Yaskawa INFORM job: SKRZYNIA_5040_0_STOPNI_2OBR.JBI

/JOB
//NAME SKRZYNIA_5040_0_STOPNI_2OBR
///FOLDERNAME 02-SKRZYNIE_JOBS
//POS
///NPOS 486,486,0,40,0,0
///TOOL 0
///POSTYPE PULSE
///PULSE
C00000=1055,-24125,84372,288,19725,204
C00001=0,-15438,65714,0,-68532,0
C00002=4718,-16587,59952,3396,-65485,-935
C00003=32997,-21499,42555,27623,-61436,21376
C00004=31759,-20688,42932,26837,-60850,21559
C00005=28987,-21156,42712,24818,-60442,22222
C00006=33447,-21964,42352,27886,-61721,21330
C00007=37687,-23357,41794,30651,-63289,20620
C00008=38979,-19018,48057,32961,-64962,20678
C00009=37261,-18075,48526,31902,-64209,20901
C00010=35830,-17198,48994,31015,-63571,21092
C00011=34080,-17614,48768,29780,-63290,21485
C00012=37261,-18075,48526,31902,-64209,20901
C00013=47373,-21912,40596,41149,-66086,26950
C00014=4718,-16587,59952,3396,-65485,-935
C00015=9265,-17323,54007,6858,-62132,-2051
C00016=8830,-16324,54489,6560,-61693,-1980
C00017=6020,-16550,54375,4472,-61664,-1348
C00018=9265,-17323,54007,6858,-62132,-2051
C00019=9252,-17290,54021,6848,-62117,-2048
C00020=9252,-17290,54021,6848,-62117,-2048
C00021=8694,-15983,54664,6467,-61548,-1957
C00022=4418,-16236,54535,3285,-61485,-993
C00023=9252,-17290,54021,6848,-62117,-2048
C00024=8708,-18333,53563,6422,-62559,-1899
C00025=8708,-18333,53563,6422,-62559,-1899
C00026=7766,-16032,54635,5782,-61526,-1748
C00027=5536,-16243,54528,4122,-61523,-1244
C00028=8708,-18333,53563,6422,-62559,-1899
C00029=8708,-18333,53563,6422,-62559,-1899
C00030=8708,-18331,53563,6422,-62556,-1899
C00031=7758,-16002,54651,5775,-61511,-1746
C00032=4943,-16221,54537,3680,-61495,-1109
C00033=30098,-19369,49260,26650,-63246,1300
C00034=73517,-47200,-15425,81407,-61841,11109
C00035=59944,-42786,-13955,78333,-53158,10478
C00036=57437,-41828,-13292,77672,-51559,10479
C00037=55365,-40827,-12885,77319,-50190,10340
C00038=53830,-41542,-13178,76508,-49301,10646
C00039=57437,-41828,-13292,77672,-51559,10479
C00040=52398,-46622,-9296,62308,-52824,5916
C00041=23564,-39822,17337,24809,-47524,-9372
C00042=10104,-46603,4759,11228,-37390,-5046
C00043=0,-52280,40443,0,6876,0
C00044=1529,-42140,58025,-5964,2417,3265
C00045=0,-52280,-4943,-1861,-42535,447
C00046=2621,-57340,-29475,1206,-23680,-711
C00047=2621,-57340,-29475,1206,-23680,-711
C00048=2622,-57337,-29476,1207,-23680,-710
C00049=2506,-56325,-29286,1041,-23045,-642
C00050=-1228,-56520,-29324,-5243,-23254,2072
C00051=2622,-57337,-29476,1207,-23680,-710
C00052=3066,-60430,-29907,1796,-25718,-952
C00053=3066,-47126,-4537,1796,-25717,-952
C00054=1150,-46289,-4389,-1134,-25181,209
C00055=1064,-44762,-4067,-1313,-24253,286
C00056=-2289,-44921,-4103,-6642,-24487,2426
C00057=-2440,-47252,-5097,-6576,-25720,2369
C00058=2574,-52173,738,1108,-22518,-664
C00059=2573,-58294,-29633,1093,-24294,-659
C00060=2321,-56024,-29231,725,-22860,-505
C00061=-1822,-56214,-29269,-6293,-23108,2531
C00062=2573,-58294,-29633,1093,-24294,-659
C00063=26763,-41451,10217,33856,-29391,24493
C00064=43270,-28616,24993,58998,-40730,16959
C00065=40951,-27396,25513,57868,-39388,17043
C00066=39074,-27880,25300,56233,-38652,17553
C00067=43270,-28616,24993,58998,-40730,16959
C00068=49158,-38250,8479,66986,-41880,13443
C00069=1817,-44984,2816,-3462,-45659,1296
C00070=1148,-56354,34370,-22,3827,-10
C00071=0,-52280,40443,0,6876,0
C00072=0,-52280,40443,0,-64237,0
C00073=12053,-46193,863,14693,-33250,-5548
C00074=7764,-43650,5766,9193,-34179,-3413
C00075=6226,-39841,6502,7870,-31713,-3015
C00076=3343,-40039,6452,4230,-31654,-1619
C00077=7764,-43650,5766,9193,-34179,-3413
C00078=7764,-43650,5766,9193,-34179,-3413
C00079=12053,-46193,863,14693,-33250,-5548
C00080=0,-52280,40443,0,6876,0
C00081=0,-52280,40443,0,6876,0
C00082=0,-52280,40443,0,6876,0
C00083=33629,-57276,-6399,46271,-24969,-2804
C00084=75493,-63502,-64712,103874,-64610,-6298
C00085=47077,-58045,-62565,110120,-45736,-10942
C00086=43793,-59800,-66982,115317,-43706,-9888
C00087=62671,-64213,-64640,104431,-56093,-7372
C00088=62671,-64213,-64640,104431,-56093,-7372
C00089=28458,-50318,6850,47420,-25887,-3347
C00090=0,-52280,40443,0,6876,0
C00091=1055,-24125,84372,288,19725,204
C00092=0,-15438,65714,0,-68532,0
C00093=0,-15438,65714,966,-70097,42926
C00094=69988,-9219,57065,61610,-82752,27767
C00095=63113,-6157,59685,58080,-79692,28271
C00096=45688,-7238,64427,40079,-74101,29444
C00097=49853,-5945,65929,43750,-75729,29302
C00098=63113,-6157,59685,58080,-79692,28271
C00099=69988,-9219,57065,61610,-82752,27767
C00100=0,-15438,65714,966,-70097,42926
C00101=0,-15438,65714,0,-68532,0
C00102=1055,-24125,84372,288,19725,204
C00103=0,-52280,40443,0,6876,0
C00104=0,-52280,40443,0,6876,0
C00105=0,-17525,61946,0,273,32004
C00106=54446,-4421,37881,-48560,57645,57448
C00107=45059,-5790,38757,-53071,45868,54447
C00108=47158,-5256,55782,-85306,41004,71351
C00109=33649,8804,54222,-37726,47106,40629
C00110=39487,-20381,-13316,-29947,69517,34787
C00111=45059,-5790,38757,-53071,45868,54447
C00112=54446,-4421,37881,-48560,57645,57448
C00113=0,-17525,61946,0,273,32004
C00114=0,-52280,40443,0,6876,0
C00115=0,-38538,66749,0,-898,0
C00116=0,-52280,40443,0,-79033,35417
C00117=46775,-35113,22190,42926,-67531,20697
C00118=52587,-26056,25345,47610,-66542,17970
C00119=45955,-25207,25003,44102,-63302,18882
C00120=46479,-26455,22189,44748,-62817,18409
C00121=53914,-29436,22058,48262,-67266,17843
C00122=46775,-35113,22190,42926,-67531,20697
C00123=0,-52280,40443,0,-79033,35417
C00124=0,-52280,40443,0,-61239,28081
C00125=53819,-14110,13758,-46164,60155,50576
C00126=48398,-14119,9451,-44868,59619,48162
C00127=40831,-18219,20924,-60631,39508,52867
C00128=25168,-7888,23888,-27338,44347,31248
C00129=48398,-14119,9451,-44868,59619,48162
C00130=63113,-6157,59685,58080,-79692,28271
C00131=47789,-6280,67353,41142,-75661,29541
C00132=46856,-5642,67903,40595,-75324,29647
C00133=49398,-5231,67705,43314,-76061,29572
C00134=31009,-27517,39857,26049,-56286,31820
C00135=0,-52280,40443,0,-61239,28081
C00136=0,-52280,40443,0,6876,0
C00137=0,-52280,40443,0,6876,0
C00138=-99253,-13690,44082,59847,13407,-31313
C00139=-87814,-12734,20141,45739,-14352,-64418
C00140=-86669,-6582,30812,41148,-16781,-62025
C00141=-85055,-5827,31548,44003,-17420,-63187
C00142=-85971,-6262,31124,42409,-17052,-62539
C00143=-86650,-5303,32069,41395,-16716,-62141
C00144=-94954,-14494,-1860,-7818,15857,-59130
C00145=-94509,-5779,9349,-537,24388,-60626
C00146=-94509,-4687,12787,-574,22838,-60605
C00147=-87106,-8124,29339,40061,-16711,-61555
C00148=-85732,-21202,11427,30682,-24763,-59235
C00149=-84150,-10929,23786,31981,-25941,-59678
C00150=-83036,-10419,24246,33504,-26268,-60308
C00151=-84150,-10929,23786,31981,-25941,-59678
C00152=-85291,-9507,25078,30650,-25411,-59154
C00153=-84150,-10929,23786,31981,-25941,-59678
C00154=-85786,-16909,14677,31743,-23900,-59790
C00155=-84150,-10498,24888,31517,-26306,-59436
C00156=-83174,-10052,25293,32841,-26587,-59984
C00157=-84150,-10498,24888,31517,-26306,-59436
C00158=-85258,-9112,26156,30226,-25800,-58928
C00159=-84150,-10498,24888,31517,-26306,-59436
C00160=-87841,-18519,13420,28367,-23534,-58339
C00161=-84150,-10465,24972,31484,-26336,-59417
C00162=-83241,-10052,25348,32714,-26598,-59924
C00163=-84150,-10465,24972,31484,-26336,-59417
C00164=-85145,-9228,26102,30329,-25881,-58963
C00165=-84150,-10465,24972,31484,-26336,-59417
C00166=-86371,-18277,13606,30568,-23951,-59265
C00167=-84345,-11688,21985,32461,-25312,-59957
C00168=-83211,-11173,22442,34044,-25650,-60618
C00169=-84345,-11688,21985,32461,-25312,-59957
C00170=-85283,-10526,23025,31366,-24861,-59525
C00171=-84345,-11688,21985,32461,-25312,-59957
C00172=-86191,-19647,12567,30467,-24278,-59187
C00173=-84345,-10877,24073,31552,-26006,-59481
C00174=-83051,-10286,24607,33321,-26381,-60213
C00175=-84345,-10877,24073,31552,-26006,-59481
C00176=-85179,-9842,25009,30582,-25619,-59100
C00177=-84345,-10877,24073,31552,-26006,-59481
C00178=-85438,-18022,14839,31140,-24818,-59429
C00179=-84247,-11820,22550,32049,-25753,-59727
C00180=-84104,-10976,23642,32111,-25899,-59738
C00181=-82990,-10465,24105,33639,-26227,-60372
C00182=-84104,-10976,23642,32111,-25899,-59738
C00183=-84898,-9998,24525,31196,-25529,-59378
C00184=-84104,-10976,23642,32111,-25899,-59738
C00185=-86610,-16845,14732,30573,-23614,-59301
C00186=-84104,-10864,23927,31990,-25993,-59674
C00187=-82824,-10273,24459,33737,-26370,-60397
C00188=-84104,-10864,23927,31990,-25993,-59674
C00189=-84789,-10021,24690,31200,-25673,-59363
C00190=-84104,-10864,23927,31990,-25993,-59674
C00191=-83806,-19585,12613,33764,-25080,-60559
C00192=-83924,-10205,25475,31619,-26533,-59453
C00193=-82780,-9675,25960,33156,-26866,-60087
C00194=-83924,-10205,25475,31619,-26533,-59453
C00195=-84478,-9530,26093,30986,-26280,-59206
C00196=-83924,-10205,25475,31619,-26533,-59453
C00197=-87149,-17993,13826,29513,-23647,-58830
C00198=-84920,-13182,20975,31162,-25481,-59361
C00199=-83711,-10572,24852,32056,-26475,-59649
C00200=-82779,-10142,25241,33309,-26748,-60166
C00201=-83711,-10572,24852,32056,-26475,-59649
C00202=-84370,-9774,25579,31305,-26170,-59356
C00203=-83711,-10572,24852,32056,-26475,-59649
C00204=-83642,-3679,42021,23358,-36761,-56118
C00205=-85886,-5975,41264,18964,-40261,-54782
C00206=-83919,-11632,22322,32811,-25616,-60079
C00207=-82884,-11162,22742,34234,-25925,-60671
C00208=-83919,-11632,22322,32811,-25616,-60079
C00209=-84723,-10654,23196,31887,-25230,-59715
C00210=-83919,-11632,22322,32811,-25616,-60079
C00211=-87348,-16035,7353,17528,-35245,-56477
C00212=-86244,-15062,8172,18754,-35315,-57058
C00213=-86244,-16649,3638,19674,-33501,-57585
C00214=-85308,-16228,3988,20718,-33648,-58082
C00215=-86244,-16649,3638,19674,-33501,-57585
C00216=-86740,-15973,4201,19194,-33277,-57362
C00217=-86244,-16649,3638,19674,-33501,-57585
C00218=-73780,-8639,20128,34258,-51705,-52097
C00219=-90711,-17528,-28778,11328,-28245,-57111
C00220=-92565,-19610,-33223,7138,-24591,-57051
C00221=-91512,-19116,-32812,8551,-24603,-57834
C00222=-92565,-19610,-33223,7138,-24591,-57051
C00223=-93003,-18716,-32476,6600,-24397,-56752
C00224=-92565,-19610,-33223,7138,-24591,-57051
C00225=-92565,-19610,-33223,7138,-24591,-57051
C00226=-95836,-54375,-51122,6031,-17685,-48210
C00227=-95836,-54375,-51122,6031,-17685,-48210
C00228=-43821,-47238,-2775,-3022,56549,-3681
C00229=-20126,-26882,59542,2406,16879,-9162
C00230=-20126,-26882,59542,2406,16879,-9162
C00231=98601,-10520,92678,4674,-40855,-9615
C00232=95537,-19831,-2695,-2933,-44471,35837
C00233=92548,-20391,-28429,-6186,-30623,55200
C00234=91429,-17018,-28974,-8057,-27827,56250
C00235=91429,-17018,-28974,-8057,-27827,56250
C00236=90371,-16495,-28521,-9286,-27856,56953
C00237=91429,-17018,-28974,-8057,-27827,56250
C00238=92033,-15799,-27911,-7415,-27588,55880
C00239=91429,-17018,-28974,-8057,-27827,56250
C00240=92548,-20391,-28429,-6186,-30623,55200
C00241=91156,-15018,-4648,-8036,-38181,54813
C00242=90585,-14766,-4428,-8565,-38201,55100
C00243=88830,-13959,-3717,-10186,-38284,55977
C00244=89897,-14456,-4157,-9202,-38230,55445
C00245=90761,-12944,-2809,-8452,-37927,55043
C00246=89897,-14456,-4157,-9202,-38230,55445
C00247=89910,-11217,67535,-9455,-58896,55399
C00248=89655,-8493,73265,-9548,-61393,54478
C00249=89910,-11217,67535,-9455,-58896,55399
C00250=85786,-16735,14816,-31782,-23869,59812
C00251=83514,-12996,17929,-35760,-24132,61552
C00252=82251,-12406,18443,-37550,-24551,62308
C00253=83514,-12996,17929,-35760,-24132,61552
C00254=84258,-12095,18717,-34917,-23742,61217
C00255=83514,-12996,17929,-35760,-24132,61552
C00256=87149,-17993,13826,-29513,-23647,58830
C00257=83118,-12818,18089,-36330,-24263,61791
C00258=81915,-12248,18589,-38020,-24666,62504
C00259=83118,-12818,18089,-36330,-24263,61791
C00260=83897,-11882,18912,-35460,-23856,61445
C00261=83118,-12818,18089,-36330,-24263,61791
C00262=83806,-19585,12613,-33764,-25080,60559
C00263=82998,-13006,17925,-36445,-24332,61826
C00264=81675,-12378,18472,-38297,-24777,62607
C00265=82998,-13006,17925,-36445,-24332,61826
C00266=83876,-11958,18841,-35466,-23874,61442
C00267=82998,-13006,17925,-36445,-24332,61826
C00268=86610,-16845,14732,-30573,-23614,59301
C00269=82493,-13239,17725,-37070,-24559,62089
C00270=81406,-12724,18174,-38578,-24928,62723
C00271=82493,-13239,17725,-37070,-24559,62089
C00272=83436,-12134,18690,-36041,-24064,61684
C00273=82493,-13239,17725,-37070,-24559,62089
C00274=84814,-16043,15376,-33312,-24093,60464
C00275=82555,-13613,17404,-36910,-24580,62015
C00276=81384,-13062,17878,-38534,-24974,62698
C00277=82555,-13613,17404,-36910,-24580,62015
C00278=83566,-12434,18427,-35805,-24047,61580
C00279=82555,-13613,17404,-36910,-24580,62015
C00280=86191,-19647,12567,-30467,-24278,59187
C00281=82500,-13648,17375,-36975,-24607,62039
C00282=81467,-13161,17792,-38413,-24955,62645
C00283=82500,-13648,17375,-36975,-24607,62039
C00284=83481,-12505,18364,-35905,-24087,61617
C00285=82500,-13648,17375,-36975,-24607,62039
C00286=86371,-18277,13606,-30568,-23951,59265
C00287=82904,-13790,17251,-36416,-24470,61808
C00288=81715,-13237,17726,-38081,-24865,62509
C00289=82904,-13790,17251,-36416,-24470,61808
C00290=83686,-12878,18037,-35556,-24055,61469
C00291=82904,-13790,17251,-36416,-24470,61808
C00292=87841,-18519,13420,-28367,-23534,58339
C00293=82748,-13879,17174,-36603,-24542,61883
C00294=81692,-13388,17594,-38077,-24893,62505
C00295=82748,-13879,17174,-36603,-24542,61883
C00296=83607,-12881,18032,-35663,-24082,61515
C00297=82748,-13879,17174,-36603,-24542,61883
C00298=85786,-16909,14677,-31743,-23900,59790
C00299=82520,-14198,16902,-36833,-24674,61972
C00300=81460,-13708,17319,-38301,-25026,62591
C00301=82520,-14198,16902,-36833,-24674,61972
C00302=83571,-12989,17938,-35691,-24113,61524
C00303=82520,-14198,16902,-36833,-24674,61972
C00304=85732,-21202,11427,-30682,-24763,59235
C00305=82398,-14365,16763,-36952,-24745,62014
C00306=81172,-13798,17245,-38643,-25153,62725
C00307=82398,-14365,16763,-36952,-24745,62014
C00308=83600,-12984,17944,-35650,-24102,61504
C00309=82398,-14365,16763,-36952,-24745,62014
C00310=83143,-16385,15097,-35497,-24760,61361
C00311=86140,-12802,12665,-93523,-10743,85795
C00312=85030,-12289,13120,-93723,-11463,85776
C00313=86140,-12802,12665,-93523,-10743,85795
C00314=86958,-11660,13681,-94506,-10238,86349
C00315=87761,-14801,10937,-92035,-9671,85255
C00316=85239,-16743,-4327,42764,21357,45785
C00317=86674,-5758,5677,19250,31526,54671
C00318=86674,-5357,7026,19593,30941,54483
C00319=94673,-11479,1830,3057,22580,57096
C00320=98660,-17899,-876,-15689,14841,63060
C00321=92405,-28594,-4465,-20793,-41,59345
C00322=85045,-36869,-4353,-28502,-22832,52282
C00323=79224,-50910,-4722,-18959,-29823,23613
C00324=0,-24029,84339,0,19981,0
C00325=3172,-24246,80980,3465,15913,689
C00326=-86563,-26985,13879,10257,-21548,-45530
C00327=-86191,-19647,12567,30467,-24278,-59187
C00328=-83221,-13587,17636,37793,-25116,-62228
C00329=-81903,-12893,15375,42337,-24108,-64400
C00330=-82005,-13000,15002,42488,-23932,-64495
C00331=-84074,-17488,11256,38660,-23649,-62784
C00332=-73679,-33270,1000,44272,-31600,-64253
C00333=-86926,-60758,23267,6576,1160,-9545
C00334=0,-52280,40443,0,6876,0
C00335=82475,-58079,26734,835,4084,4444
C00336=97932,-26840,7691,8784,-23444,42538
C00337=87166,-16607,16322,-25365,-24201,56345
C00338=84591,-11487,21632,-29278,-24784,58002
C00339=84698,-11389,22004,-28939,-24910,57841
C00340=85100,-26994,10417,-24982,-28140,55821
C00341=0,-52280,40443,0,6876,0
C00342=0,-52280,40443,0,6876,0
C00343=-90140,-60305,18108,-2708,1721,-7625
C00344=-95594,-27428,6866,-4663,-19832,-42154
C00345=-98688,-13767,16447,-18366,-10080,-35766
C00346=-95535,2380,25473,239,27557,-47214
C00347=-90841,2528,33450,-5594,22315,-43657
C00348=-95534,12422,45149,295,21566,-47242
C00349=-99268,-13088,27343,-18620,-14105,-35021
C00350=-88464,-60269,18234,-16733,1666,-1052
C00351=0,-52280,40443,0,6876,0
C00352=84259,-57935,27522,-3761,3673,6310
C00353=86507,-39672,4297,-27618,-16640,46340
C00354=73669,-37119,-20783,-92053,-19719,85232
C00355=92187,-27573,7158,-33072,-13361,58684
C00356=94920,-15931,-8336,1617,33944,36739
C00357=93066,-3679,7807,-1859,41451,36204
C00358=97249,5774,18161,-4516,41609,38146
C00359=100487,-9453,-1206,-10413,41328,41147
C00360=96250,-19428,-8283,-4838,27297,37910
C00361=86507,-39672,4297,-27618,-16640,46340
C00362=84259,-57935,27522,-3761,3673,6310
C00363=0,-52280,40443,0,6876,0
C00364=0,-27933,77061,0,20812,0
C00365=0,-27933,77061,0,20812,0
C00366=0,-52280,40443,0,6876,0
C00367=-91970,-60791,14435,-3343,512,-9412
C00368=-98647,-24138,10005,-11519,-21203,-39749
C00369=-99883,-13980,22886,-11640,-25090,-40341
C00370=-99702,-9154,61728,-1148,-61809,-40243
C00371=-84328,-13042,29707,23458,-33731,-54641
C00372=-83101,-4179,39208,25894,-34785,-55667
C00373=-82881,-4330,38692,26392,-34479,-55866
C00374=-76259,-18287,26646,31659,-38322,-57579
C00375=-89741,-28009,12101,4461,-28076,-46404
C00376=-91970,-60791,14435,-3343,512,-9412
C00377=0,-52280,40443,0,6876,0
C00378=91083,-60784,14823,-9043,-825,15173
C00379=83869,-19403,12921,-33769,-24740,60260
C00380=83869,-19403,12921,-33769,-24740,60260
C00381=83932,-19538,53415,-33663,-71112,60249
C00382=83932,-19538,53415,-33663,-71112,60249
C00383=82480,-12247,21118,-35440,-26416,60009
C00384=82194,-11433,19802,-37650,-25323,61125
C00385=81904,-9374,24711,-35791,-26879,60109
C00386=79790,-20261,14917,-36681,-28829,60258
C00387=76554,-29711,-1870,-46042,-25952,65654
C00388=91083,-60784,14823,-9043,-825,15173
C00389=0,-52280,40443,0,6876,0
C00390=-91526,-60598,16699,7584,176,-13289
C00391=-81382,-25890,9219,35455,-25500,-59095
C00392=-86453,-20958,12525,30076,-22568,-57089
C00393=-86589,-16097,16237,31250,-21582,-57704
C00394=-98933,-11298,20505,-13970,-18736,-37953
C00395=-98281,-10965,21163,-11559,-18548,-39330
C00396=-85424,-18472,14402,34409,-22969,-58895
C00397=-74746,-27148,8488,44263,-29128,-62418
C00398=-81326,-27507,8265,35533,-26282,-59001
C00399=-91415,-60262,16631,7870,-73,-13734
C00400=24,-24029,84339,7,19981,5
C00401=100404,-52373,45687,-1822,14816,-5144
C00402=75939,-26469,7919,-40869,-29645,63133
C00403=81882,-22565,10470,-35355,-26404,61107
C00404=82801,-12246,21732,-34208,-26055,60642
C00405=92083,-10555,23625,-8209,-22171,49629
C00406=97182,-9584,26244,6847,-23189,43246
C00407=77262,-23244,14300,-38922,-31295,61912
C00408=78410,-30298,-3216,-47287,-24876,66197
C00409=90612,-54995,-11460,93167,-17168,-8155
C00410=568,-24029,84339,168,19981,112
C00411=-91970,-60791,14435,-3343,512,-9412
C00412=-98991,-22833,11519,-12824,-17638,-36336
C00413=-86376,-13627,18436,38326,-18406,-58533
C00414=-85581,-10814,20279,41280,-18093,-59893
C00415=-85551,-10406,21021,40925,-18257,-59713
C00416=-86274,-24518,9978,34497,-20333,-56613
C00417=-91684,-53777,2301,20525,-9313,-33684
C00418=-67305,-55044,34987,1504,5690,-2468
C00419=0,-52280,40443,0,6876,0
C00420=77036,-56616,31288,-2531,4707,4197
C00421=84359,-28321,8817,-32860,-20485,54199
C00422=81156,-16932,14874,-39538,-26422,62851
C00423=93122,-15135,13007,-5735,-18111,48773
C00424=90767,-14192,15510,-13532,-19632,52035
C00425=77970,-27630,4721,-41834,-28549,63607
C00426=81111,-35571,7141,-33980,-21909,52006
C00427=82626,-57814,28323,-4146,3364,6346
C00428=0,-52280,40443,0,6876,0
C00429=0,-28135,76691,0,20839,0
C00430=0,-28135,76691,0,20839,0
C00431=-45332,-39712,59352,-1730,18713,2903
C00432=-94065,-8316,59352,-1730,-37754,-40387
C00433=-100331,-14895,33931,-8215,-36518,-40227
C00434=-98931,-8578,39429,-6260,-48307,-43744
C00435=-100336,-4176,46216,-7600,-55875,-44633
C00436=-93952,8947,73671,995,-68520,-43850
C00437=-98791,-3170,32594,-4861,-60761,-43748
C00438=-98617,4601,38180,-4851,-58752,-43714
C00439=-98607,-12593,-18438,-7609,-32838,-41877
C00440=-98632,-14188,-28321,-9032,-27293,-41100
C00441=-99605,-15546,-21493,-8548,-33053,-41326
C00442=-100467,-8208,-2562,-8095,-44661,-42156
C00443=-93952,8947,73671,995,-68520,-43850
C00444=-88754,54,62805,4404,-67858,-45120
C00445=-100222,-4532,45667,-7492,-55263,-44561
C00446=-100331,-14895,33931,-8215,-36518,-40227
C00447=-94065,-8316,59352,-1730,-37754,-40387
C00448=-45544,-32973,71870,-2133,15168,3033
C00449=0,-28135,76691,0,20839,0
C00450=54178,-17846,77779,596,-29686,20997
C00451=54178,-17846,77779,596,-29686,20997
C00452=99462,-18987,75418,611,-28919,20989
C00453=98707,-9390,78674,1080,-71212,38250
C00454=98768,-5182,41096,1808,-44974,38308
C00455=100431,1771,51615,3823,-56746,39115
C00456=97953,-6621,17555,2289,-50176,39420
C00457=95834,-5353,18817,760,-50052,40242
C00458=86453,-3910,18511,-13431,-48443,44868
C00459=88887,-11110,-8515,-11527,-36861,46615
C00460=88808,-13839,-20865,-13699,-30585,47852
C00461=91485,-7261,12020,-7409,-47660,44146
C00462=97953,-6621,17555,2289,-50176,39420
C00463=100431,1771,51615,3823,-56746,39115
C00464=98768,-5182,41096,1808,-44974,38308
C00465=98707,-9390,78674,1080,-71212,38250
C00466=0,-28135,76691,0,20839,0
C00467=0,-28135,76691,0,20839,0
C00468=-91526,-60598,16699,7584,176,-13289
C00469=-81382,-25890,9219,35455,-25500,-59095
C00470=-81382,-25890,9219,35455,-25500,-59095
C00471=-85509,-13950,19358,32213,-22393,-58041
C00472=-96341,-12086,19487,-5053,-17846,-42145
C00473=-97523,-9822,24708,-8570,-19966,-40659
C00474=-84656,-25369,12054,31249,-26195,-57129
C00475=-82652,-57346,29982,2770,3944,-5064
C00476=0,-52280,40443,0,6876,0
C00477=60653,-54633,35892,-1212,5841,2035
C00478=77942,-28227,6869,-38010,-29303,61907
C00479=82500,-13648,17375,-36975,-24607,62039
C00480=80731,-11587,18684,-41654,-25449,63953
C00481=80409,-10373,22284,-40214,-26848,63104
C00482=64389,-31987,5108,-50419,-37074,66126
C00483=60653,-54633,35892,-1212,5841,2035
C00484=0,-52280,40443,0,6876,0
C00485=0,-28167,76633,0,20843,0
BC00000=413138
BC00001=413138
BC00002=295997
BC00003=264574
BC00004=264574
BC00005=264574
BC00006=264574
BC00007=233852
BC00008=284288
BC00009=284288
BC00010=284288
BC00011=284288
BC00012=284288
BC00013=356545
BC00014=388163
BC00015=356740
BC00016=356740
BC00017=356740
BC00018=356740
BC00019=407176
BC00020=407176
BC00021=407176
BC00022=407176
BC00023=413370
BC00024=479433
BC00025=479433
BC00026=479433
BC00027=479433
BC00028=479433
BC00029=534201
BC00030=534204
BC00031=534204
BC00032=534204
BC00033=534204
BC00034=538468
BC00035=598406
BC00036=603654
BC00037=603654
BC00038=603654
BC00039=603654
BC00040=590790
BC00041=556978
BC00042=522422
BC00043=507734
BC00044=671734
BC00045=689202
BC00046=689202
BC00047=689202
BC00048=689201
BC00049=689201
BC00050=689201
BC00051=689201
BC00052=689202
BC00053=726463
BC00054=726463
BC00055=726463
BC00056=726463
BC00057=727112
BC00058=762991
BC00059=811128
BC00060=811128
BC00061=811128
BC00062=811128
BC00063=808294
BC00064=808294
BC00065=808294
BC00066=808294
BC00067=808294
BC00068=808294
BC00069=823841
BC00070=719909
BC00071=755227
BC00072=899666
BC00073=899666
BC00074=899666
BC00075=899666
BC00076=899666
BC00077=899666
BC00078=899666
BC00079=899666
BC00080=838173
BC00081=727925
BC00082=734552
BC00083=734552
BC00084=750834
BC00085=750837
BC00086=812765
BC00087=812765
BC00088=760768
BC00089=744267
BC00090=744267
BC00091=413138
BC00092=413138
BC00093=413138
BC00094=408626
BC00095=408626
BC00096=408753
BC00097=347392
BC00098=408626
BC00099=408626
BC00100=413138
BC00101=413138
BC00102=413138
BC00103=838173
BC00104=697681
BC00105=697681
BC00106=722402
BC00107=758324
BC00108=766520
BC00109=807455
BC00110=807455
BC00111=758324
BC00112=733666
BC00113=677371
BC00114=697681
BC00115=507816
BC00116=507816
BC00117=552804
BC00118=552804
BC00119=551170
BC00120=492063
BC00121=491979
BC00122=552804
BC00123=507816
BC00124=507816
BC00125=507816
BC00126=531288
BC00127=531293
BC00128=576030
BC00129=531288
BC00130=285738
BC00131=285865
BC00132=285441
BC00133=256782
BC00134=325752
BC00135=507816
BC00136=507816
BC00137=818250
BC00138=831179
BC00139=948272
BC00140=948272
BC00141=948272
BC00142=948272
BC00143=948272
BC00144=948272
BC00145=948272
BC00146=948272
BC00147=948272
BC00148=902188
BC00149=895372
BC00150=895372
BC00151=895372
BC00152=895372
BC00153=895372
BC00154=840744
BC00155=840744
BC00156=840744
BC00157=840744
BC00158=840744
BC00159=840744
BC00160=779300
BC00161=771332
BC00162=771332
BC00163=771332
BC00164=771332
BC00165=771332
BC00166=717855
BC00167=717855
BC00168=717855
BC00169=717855
BC00170=717855
BC00171=717855
BC00172=656405
BC00173=649173
BC00174=649173
BC00175=649173
BC00176=649173
BC00177=649173
BC00178=594961
BC00179=594961
BC00180=594961
BC00181=594961
BC00182=594961
BC00183=594961
BC00184=594961
BC00185=533517
BC00186=525229
BC00187=525229
BC00188=525229
BC00189=525229
BC00190=525229
BC00191=472073
BC00192=472073
BC00193=472073
BC00194=472073
BC00195=472073
BC00196=472073
BC00197=410629
BC00198=405662
BC00199=402968
BC00200=402968
BC00201=402968
BC00202=402968
BC00203=402968
BC00204=402968
BC00205=349186
BC00206=349186
BC00207=349186
BC00208=349186
BC00209=349186
BC00210=349186
BC00211=336469
BC00212=336469
BC00213=336469
BC00214=336469
BC00215=336469
BC00216=336469
BC00217=336469
BC00218=367602
BC00219=367601
BC00220=367601
BC00221=367601
BC00222=367601
BC00223=367601
BC00224=367601
BC00225=425303
BC00226=425303
BC00227=514953
BC00228=463119
BC00229=419862
BC00230=484962
BC00231=484962
BC00232=395463
BC00233=369502
BC00234=369502
BC00235=369502
BC00236=369502
BC00237=369502
BC00238=369502
BC00239=369502
BC00240=369502
BC00241=368885
BC00242=368885
BC00243=368885
BC00244=368885
BC00245=368885
BC00246=368885
BC00247=419064
BC00248=419064
BC00249=366918
BC00250=349186
BC00251=353241
BC00252=353241
BC00253=353241
BC00254=353241
BC00255=353241
BC00256=410629
BC00257=409135
BC00258=409135
BC00259=409135
BC00260=409135
BC00261=409135
BC00262=472073
BC00263=476126
BC00264=476126
BC00265=476126
BC00266=476126
BC00267=476126
BC00268=533517
BC00269=532644
BC00270=532644
BC00271=532644
BC00272=532644
BC00273=532644
BC00274=594961
BC00275=599988
BC00276=599988
BC00277=599988
BC00278=599988
BC00279=599988
BC00280=656405
BC00281=653254
BC00282=653254
BC00283=653254
BC00284=653254
BC00285=653254
BC00286=717855
BC00287=721570
BC00288=721570
BC00289=721570
BC00290=721570
BC00291=721570
BC00292=779300
BC00293=777963
BC00294=777963
BC00295=777963
BC00296=777963
BC00297=777963
BC00298=840744
BC00299=843810
BC00300=843810
BC00301=843810
BC00302=843810
BC00303=843810
BC00304=902188
BC00305=900128
BC00306=900128
BC00307=900128
BC00308=900128
BC00309=900128
BC00310=900128
BC00311=950128
BC00312=950128
BC00313=950128
BC00314=950128
BC00315=950128
BC00316=950128
BC00317=950128
BC00318=950128
BC00319=950128
BC00320=944131
BC00321=934334
BC00322=916143
BC00323=861901
BC00324=769966
BC00325=716686
BC00326=679663
BC00327=721442
BC00328=721442
BC00329=721439
BC00330=781482
BC00331=781888
BC00332=781888
BC00333=781888
BC00334=781888
BC00335=768943
BC00336=718475
BC00337=718475
BC00338=718475
BC00339=778313
BC00340=778313
BC00341=717855
BC00342=792672
BC00343=792672
BC00344=917473
BC00345=917473
BC00346=925953
BC00347=925953
BC00348=925953
BC00349=919477
BC00350=761950
BC00351=761950
BC00352=761950
BC00353=856724
BC00354=925542
BC00355=925542
BC00356=942328
BC00357=941076
BC00358=941460
BC00359=925542
BC00360=925542
BC00361=887446
BC00362=792672
BC00363=792672
BC00364=700249
BC00365=546214
BC00366=546214
BC00367=546211
BC00368=546211
BC00369=406776
BC00370=406776
BC00371=352261
BC00372=346119
BC00373=406266
BC00374=406266
BC00375=491556
BC00376=546211
BC00377=546214
BC00378=546214
BC00379=507604
BC00380=410782
BC00381=429690
BC00382=375447
BC00383=350474
BC00384=350474
BC00385=408658
BC00386=408658
BC00387=507604
BC00388=546214
BC00389=546214
BC00390=516757
BC00391=591809
BC00392=591809
BC00393=591809
BC00394=591183
BC00395=650353
BC00396=650538
BC00397=650538
BC00398=584003
BC00399=515801
BC00400=520018
BC00401=520018
BC00402=590597
BC00403=593080
BC00404=593080
BC00405=593080
BC00406=652456
BC00407=652559
BC00408=594501
BC00409=537666
BC00410=433888
BC00411=546211
BC00412=830322
BC00413=830322
BC00414=830322
BC00415=890247
BC00416=890396
BC00417=798848
BC00418=798848
BC00419=798848
BC00420=798848
BC00421=832296
BC00422=845010
BC00423=845010
BC00424=904605
BC00425=904704
BC00426=818840
BC00427=818839
BC00428=818839
BC00429=526967
BC00430=334612
BC00431=334612
BC00432=334612
BC00433=350464
BC00434=350464
BC00435=359337
BC00436=359337
BC00437=359337
BC00438=359337
BC00439=359337
BC00440=359337
BC00441=359337
BC00442=359337
BC00443=359337
BC00444=359337
BC00445=358620
BC00446=350464
BC00447=334612
BC00448=334612
BC00449=334612
BC00450=334613
BC00451=501279
BC00452=501279
BC00453=334612
BC00454=334610
BC00455=349510
BC00456=365935
BC00457=365935
BC00458=365934
BC00459=348430
BC00460=348430
BC00461=348430
BC00462=365935
BC00463=349510
BC00464=334610
BC00465=334612
BC00466=334612
BC00467=512789
BC00468=516757
BC00469=526627
BC00470=466969
BC00471=466969
BC00472=466969
BC00473=524647
BC00474=525745
BC00475=525745
BC00476=525745
BC00477=525745
BC00478=473911
BC00479=473911
BC00480=473911
BC00481=532824
BC00482=533743
BC00483=525745
BC00484=525745
BC00485=525747
///POSTYPE BASE
///RECTAN
///RCONF 0,0,0,0,0,0,0,0,0,0,0,0,0,0,0,0,0,0,0,0,0,0,0,0
P00006=-2.449,0.031,8.825,0.0000,0.0000,0.0000
P00057=0.000,0.000,2.000,0.0000,0.0000,0.0000
///RCONF 1,0,0,0,0,0,0,0,0,0,0,0,0,0,0,0,0,0,0,0,0,0,0,0
P00097=0.043,-1.896,1.568,0.0000,0.0000,0.0000
P00098=-0.089,-2.467,4.059,0.0000,0.0000,0.0000
P00099=0.011,-2.380,1.226,0.0000,0.0000,0.0000
P00100=-0.081,2.558,4.482,0.0000,0.0000,0.0000
P00101=0.030,-2.286,2.993,0.0000,0.0000,0.0000
P00102=-0.005,-1.108,1.644,0.0000,0.0000,0.0000
P00103=-0.094,-3.400,4.200,0.0000,0.0000,0.0000
P00104=0.043,-2.127,5.826,0.0000,0.0000,0.0000
P00105=-0.043,0.662,5.286,0.0000,0.0000,0.0000
P00106=-0.018,-2.519,0.237,0.0000,0.0000,0.0000
P00107=-0.008,-4.537,-4.500,0.0000,0.0000,0.0000
P00108=0.014,-3.040,2.637,0.0000,0.0000,0.0000
///RCONF 0,0,0,0,0,0,0,0,0,0,0,0,0,0,0,0,0,0,0,0,0,0,0,0
P00299=-3.815,-1.565,6.918,0.0000,0.0000,0.0000
P00301=0.005,-4.708,-4.628,0.0000,0.0000,0.0000
P00302=0.052,-2.937,-4.426,0.0000,0.0000,0.0000
P00303=-0.004,-1.437,-4.584,0.0000,0.0000,0.0000
P00304=0.028,-1.666,-4.234,0.0000,0.0000,0.0000
P00305=-0.003,-1.920,-3.501,0.0000,0.0000,0.0000
P00306=0.015,-2.252,-3.054,0.0000,0.0000,0.0000
P00307=0.019,-2.151,-5.077,0.0000,0.0000,0.0000
P00308=-0.003,-2.092,-4.888,0.0000,0.0000,0.0000
P00309=-0.040,-2.205,-4.992,0.0000,0.0000,0.0000
P00310=-0.006,-2.490,-5.925,0.0000,0.0000,0.0000
P00311=-0.007,-2.079,-5.307,0.0000,0.0000,0.0000
P00312=-0.032,2.202,-7.632,0.0000,0.0000,0.0000
///RCONF 1,0,0,0,0,0,0,0,0,0,0,0,0,0,0,0,0,0,0,0,0,0,0,0
P00349=0.060,0.167,-1.133,0.0000,0.0000,0.0000
///RCONF 0,0,0,0,0,0,0,0,0,0,0,0,0,0,0,0,0,0,0,0,0,0,0,0
P00350=11.519,-0.008,1.149,0.0000,0.0000,0.0000
P00351=13.563,-0.027,-0.653,0.0000,0.0000,0.0000
P00352=13.252,-0.027,-0.827,0.0000,0.0000,0.0000
P00353=10.971,-0.082,0.776,0.0000,0.0000,0.0000
P00354=-0.024,2.508,-1.824,0.0000,0.0000,0.0000
P00355=-0.001,2.528,-1.131,0.0000,0.0000,0.0000
P00356=-0.034,2.921,-0.262,0.0000,0.0000,0.0000
P00357=0.003,3.386,-0.091,0.0000,0.0000,0.0000
P00358=0.014,3.037,-0.020,0.0000,0.0000,0.0000
P00359=-0.005,2.731,0.912,0.0000,0.0000,0.0000
P00360=-0.011,3.412,0.438,0.0000,0.0000,0.0000
P00361=0.018,3.050,1.253,0.0000,0.0000,0.0000
//INST
///DATE 2025/06/06 12:09
///ATTR SC,RW
///GROUP1 RB1,BS1
NOP
CALL JOB:MOVE_INTO_TUNNEL
SFTOF
'------------------------
'------------------------
'SPOINA SRODEK DOL
'------------------------
'------------------------
MOVJ C00000 BC00000 VJ=10.00
MOVJ C00001 BC00001 VJ=30.00
'------------------------
'W38 P
'------------------------
'TEST
'------------------------
'PODLOGA_BEZ_ROZPORKI
'------------------------
'TEST
MOVL C00002 BC00002 V=166.7
MOVL C00003 BC00003 V=166.7 PL=0
REFP 3 C00004 BC00004
CALL JOB:SEARCH-R1
IMOV P0057 V=23.0
SET P0097 P0006
SFTON P0097
REFP 3 C00005 BC00005
CALL JOB:SEARCH-R1
SET P0097 P0006
SFTON P0097
MOVL C00006 BC00006 V=166.7 PL=0
SFTOF
COMM MOVL C00007 BC00007 V=333.3
MOVL C00008 BC00008 V=333.3
MOVL C00009 BC00009 V=166.7 PL=0
REFP 3 C00010 BC00010
CALL JOB:SEARCH-R1
IMOV P0057 V=23.0
SET P0098 P0006
SFTON P0098
REFP 3 C00011 BC00011
CALL JOB:SEARCH-R1
SET P0098 P0006
SFTON P0098
MOVL C00012 BC00012 V=166.7 PL=0
'TEST
SFTOF
MOVJ C00013 BC00013 VJ=20.00
MOVL C00014 BC00014 V=166.7
MOVL C00015 BC00015 V=133.3 PL=0
REFP 3 C00016 BC00016
CALL JOB:SEARCH-R1
IMOV P0057 V=23.0
SET P0099 P0006
SFTON P0099
REFP 3 C00017 BC00017
CALL JOB:SEARCH-R1
SET P0099 P0006
SFTON P0099
MOVL C00018 BC00018 V=66.7 PL=0
'TEST
SFTOF
MOVJ C00019 BC00019 VJ=20.00
'------------------------
'W38 L
'------------------------
'TEST
MOVL C00020 BC00020 V=66.7 PL=0
REFP 3 C00021 BC00021
CALL JOB:SEARCH-R1
IMOV P0057 V=23.0
SET P0100 P0006
SFTON P0100
REFP 3 C00022 BC00022
CALL JOB:SEARCH-R1
SET P0100 P0006
SFTON P0100
MOVL C00023 BC00023 V=66.7 PL=0
'TEST
SFTOF
MOVJ C00024 BC00024 VJ=20.00
'------------------------
'W45 P
'------------------------
MOVL C00025 BC00025 V=66.7 PL=0
REFP 3 C00026 BC00026
CALL JOB:SEARCH-R1
IMOV P0057 V=23.0
SET P0101 P0006
SFTON P0101
REFP 3 C00027 BC00027
CALL JOB:SEARCH-R1
SET P0101 P0006
SFTON P0101
MOVL C00028 BC00028 V=66.7 PL=0
'TEST
SFTOF
MOVJ C00029 BC00029 VJ=20.00
'------------------------
'W45 L
'------------------------
MOVL C00030 BC00030 V=66.7 PL=0
REFP 3 C00031 BC00031
CALL JOB:SEARCH-R1
IMOV P0057 V=23.0
SET P0102 P0006
SFTON P0102
REFP 3 C00032 BC00032
CALL JOB:SEARCH-R1
SET P0102 P0006
SFTON P0102
MOVL C00033 BC00033 V=66.7 PL=0
MOVJ C00034 BC00034 VJ=20.00
'TEST
SFTOF
MOVJ C00035 BC00035 VJ=20.00
'------------------------
'W48 P
'------------------------
'TEST
MOVL C00036 BC00036 V=166.7 PL=0
REFP 3 C00037 BC00037
CALL JOB:SEARCH-R1
IMOV P0057 V=23.0
SET P0103 P0006
SFTON P0103
REFP 3 C00038 BC00038
CALL JOB:SEARCH-R1
SET P0103 P0006
SFTON P0103
MOVL C00039 BC00039 V=166.7 PL=0
'TEST
SFTOF
MOVJ C00040 BC00040 VJ=20.00
MOVJ C00041 BC00041 VJ=10.00
MOVJ C00042 BC00042 VJ=30.00
MOVJ C00043 BC00043 VJ=30.00
MOVJ C00044 BC00044 VJ=30.00
MOVJ C00045 BC00045 VJ=20.00
MOVJ C00046 BC00046 VJ=10.00
MOVL C00047 BC00047 V=250.0
'------------------------
'W48 L
'------------------------
SFTOF
MOVL C00048 BC00048 V=66.7 PL=0
REFP 3 C00049 BC00049
CALL JOB:SEARCH-R1
IMOV P0057 V=23.0
SET P0104 P0006
SFTON P0104
REFP 3 C00050 BC00050
CALL JOB:SEARCH-R1
SET P0104 P0006
SFTON P0104
MOVL C00051 BC00051 V=66.7 PL=0
SFTOF
MOVL C00052 BC00052 V=66.7
MOVJ C00053 BC00053 VJ=20.00
'------------------------
'W36 P
'------------------------
MOVL C00054 BC00054 V=66.7 PL=0
REFP 3 C00055 BC00055
CALL JOB:SEARCH-R1
IMOV P0057 V=23.0
SET P0105 P0006
SFTON P0105
REFP 3 C00056 BC00056
CALL JOB:SEARCH-R1
SET P0105 P0006
SFTON P0105
MOVL C00057 BC00057 V=66.7 PL=0
'TEST
SFTOF
MOVJ C00058 BC00058 VJ=20.00
'------------------------
'W36 L
'------------------------
MOVL C00059 BC00059 V=66.7 PL=0
REFP 3 C00060 BC00060
CALL JOB:SEARCH-R1
IMOV P0057 V=23.0
SET P0106 P0006
SFTON P0106
REFP 3 C00061 BC00061
CALL JOB:SEARCH-R1
SET P0106 P0006
SFTON P0106
MOVL C00062 BC00062 V=250.0 PL=0
'TEST
MOVJ C00063 BC00063 VJ=20.00
SFTOF
'------------------------
'W44 P
'------------------------
'TEST
MOVL C00064 BC00064 V=66.7 PL=0
REFP 3 C00065 BC00065
CALL JOB:SEARCH-R1
IMOV P0057 V=23.0
SET P0107 P0006
SFTON P0107
REFP 3 C00066 BC00066
CALL JOB:SEARCH-R1
SET P0107 P0006
SFTON P0107
MOVL C00067 BC00067 V=250.0 PL=0
'TEST
SFTOF
MOVJ C00068 BC00068 VJ=20.00
MOVJ C00069 BC00069 VJ=25.00
MOVJ C00070 BC00070 VJ=25.00
MOVJ C00071 BC00071 VJ=25.00
MOVJ C00072 BC00072 VJ=30.00
MOVJ C00073 BC00073 VJ=25.00
'------------------------
'W44 L
'------------------------
'TEST
MOVL C00074 BC00074 V=66.7 PL=0
REFP 3 C00075 BC00075
CALL JOB:SEARCH-R1
IMOV P0057 V=23.0
SET P0108 P0006
SFTON P0108
REFP 3 C00076 BC00076
CALL JOB:SEARCH-R1
SET P0108 P0006
SFTON P0108
MOVL C00077 BC00077 V=250.0 PL=0
'TEST
SFTOF
MOVL C00078 BC00078 V=150.0
MOVJ C00079 BC00079 VJ=10.00
CALL JOB:FRONT_SEARCH_0ST-2_5040_V2
MOVJ C00080 BC00080 VJ=30.00
MOVJ C00081 BC00081 VJ=40.00
'WELD
'WELD
MOVJ C00082 BC00082 VJ=10.00
MOVJ C00083 BC00083 VJ=10.00
'**********************
'W36
'**********************
MOVL C00084 BC00084 V=500.0
SFTON P0105
MOVL C00085 BC00085 V=66.7 PL=0
SFTOF
MACRO1 MJ#(0) ARGF9
ARCON
SFTON P0106
MOVL C00086 BC00086 V=11.7
ARCOF
SFTOF
MOVJ C00087 BC00087 VJ=20.00
MOVJ C00088 BC00088 VJ=20.00
MOVJ C00089 BC00089 VJ=20.00
MOVJ C00090 BC00090 VJ=20.00
MOVJ C00091 BC00091 VJ=30.00
MOVJ C00092 BC00092 VJ=20.00
MOVJ C00093 BC00093 VJ=20.00
MOVJ C00094 BC00094 VJ=20.00
'**********************
'W38
'**********************
MOVL C00095 BC00095 V=500.0
SFTON P0100
MOVL C00096 BC00096 V=166.7 PL=0
SFTOF
ARCON
SFTON P0099
MOVL C00097 BC00097 V=11.7
ARCOF
SFTOF
'DODANE
MOVL C00098 BC00098 V=500.0
MOVJ C00099 BC00099 VJ=10.00
MOVJ C00100 BC00100 VJ=20.00
MOVJ C00101 BC00101 VJ=20.00
MOVJ C00102 BC00102 VJ=30.00
MOVJ C00103 BC00103 VJ=40.00
CALL JOB:FRONT_WELD_0ST-2_5040_V2
'**********************
'W44
'**********************
MOVJ C00104 BC00104 VJ=30.00
MOVJ C00105 BC00105 VJ=20.00
MOVJ C00106 BC00106 VJ=20.00
MOVL C00107 BC00107 V=500.0
SFTON P0107
MOVL C00108 BC00108 V=100.0 PL=0
SFTOF
MACRO1 MJ#(0) ARGF9
ARCON
SFTON P0108
MOVL C00109 BC00109 V=10.0
ARCOF
SFTOF
MOVL C00110 BC00110 V=333.3
MOVL C00111 BC00111 V=500.0
MOVJ C00112 BC00112 VJ=20.00
MOVJ C00113 BC00113 VJ=20.00
MOVJ C00114 BC00114 VJ=30.00
'**********************
'DODATEK
'**********************
MOVJ C00115 BC00115 VJ=30.00
MOVJ C00116 BC00116 VJ=20.00
MOVJ C00117 BC00117 VJ=20.00
MACRO1 MJ#(0) ARGF9
MOVL C00118 BC00118 V=500.0
SFTON P0102
MOVL C00119 BC00119 V=166.7 PL=0
SFTOF
ARCON
SFTON P0101
MOVL C00120 BC00120 V=11.7
ARCOF
SFTOF
MOVL C00121 BC00121 V=500.0
MOVJ C00122 BC00122 VJ=20.00
MOVJ C00123 BC00123 VJ=30.00
'**********************
'W48
'**********************
MOVJ C00124 BC00124 VJ=30.00
MOVJ C00125 BC00125 VJ=10.00
MOVJ C00126 BC00126 VJ=20.00
SFTON P0103
MOVL C00127 BC00127 V=166.7 PL=0
SFTOF
ARCON
SFTON P0104
MOVL C00128 BC00128 V=10.0
ARCOF
SFTOF
MOVL C00129 BC00129 V=500.0
'**********************
'SPOINA_PODLOGA_BRAK_ROZP
'**********************
MOVL C00130 BC00130 V=500.0
MOVL C00131 BC00131 V=500.0
SFTON P0098
MOVL C00132 BC00132 V=166.7 PL=0
SFTOF
ARCON
SFTON P0097
MOVL C00133 BC00133 V=11.3
ARCOF
MOVL C00134 BC00134 V=333.3
SFTOF
'DODANE
MOVJ C00135 BC00135 VJ=20.00
MOVJ C00136 BC00136 VJ=30.00
CALL JOB:MOVE_OUT_OF_TUNNEL
CALL JOB:CLEAN-R1
CALL JOB:MOVE_INTO_TUNNEL
MOVJ C00137 BC00137 VJ=30.00 PL=0
'------------------------
'------------------------
'PRAWA STRONA PROFIL GORA
'------------------------
'------------------------
MOVJ C00138 BC00138 VJ=20.00
MOVJ C00139 BC00139 VJ=20.00
MOVL C00140 BC00140 V=166.7 PL=0
REFP 3 C00141 BC00141
CALL JOB:SEARCH-R1
SET P0299 P0006
SFTON P0299
MOVL C00142 BC00142 V=66.7 PL=0
REFP 3 C00143 BC00143
CALL JOB:SEARCH-R1
SET P0299 P0006
SFTON P0299
MOVL C00144 BC00144 V=83.3
MOVL C00145 BC00145 V=166.7 PL=0
REFP 3 C00146 BC00146
CALL JOB:SEARCH-R1
SET P0299 P0006
SFTON P0299
MOVL C00147 BC00147 V=250.0 PL=0
SFTOF
MOVJ C00148 BC00148 VJ=30.00
MOVL C00149 BC00149 V=166.7 PL=0
REFP 3 C00150 BC00150
CALL JOB:SEARCH-R1
SET P0301 P0006
SFTON P0301
MOVL C00151 BC00151 V=66.7 PL=0
REFP 3 C00152 BC00152
CALL JOB:SEARCH-R1
SET P0301 P0006
SFTON P0301
MOVL C00153 BC00153 V=66.7 PL=0
SFTOF
'------------------------
'W54A P
'------------------------
SFTOF
MOVJ C00154 BC00154 VJ=30.00
MOVL C00155 BC00155 V=133.3 PL=0
REFP 3 C00156 BC00156
CALL JOB:SEARCH-R1
SET P0302 P0006
SFTON P0302
MOVL C00157 BC00157 V=66.7 PL=0
REFP 3 C00158 BC00158
CALL JOB:SEARCH-R1
SET P0302 P0006
SFTON P0302
MOVL C00159 BC00159 V=66.7 PL=0
SFTOF
'------------------------
'W50A L
'------------------------
SFTOF
MOVJ C00160 BC00160 VJ=30.00
MOVL C00161 BC00161 V=133.3 PL=0
REFP 3 C00162 BC00162
CALL JOB:SEARCH-R1
SET P0303 P0006
SFTON P0303
MOVL C00163 BC00163 V=66.7 PL=0
REFP 3 C00164 BC00164
CALL JOB:SEARCH-R1
SET P0303 P0006
SFTON P0303
MOVL C00165 BC00165 V=66.7 PL=0
SFTOF
'------------------------
'W50A P
'------------------------
SFTOF
MOVJ C00166 BC00166 VJ=30.00
MOVL C00167 BC00167 V=133.3 PL=0
REFP 3 C00168 BC00168
CALL JOB:SEARCH-R1
SET P0304 P0006
SFTON P0304
MOVL C00169 BC00169 V=66.7 PL=0
REFP 3 C00170 BC00170
CALL JOB:SEARCH-R1
SET P0304 P0006
SFTON P0304
MOVL C00171 BC00171 V=66.7 PL=0
SFTOF
'------------------------
'W53A L
'------------------------
SFTOF
MOVJ C00172 BC00172 VJ=30.00
MOVL C00173 BC00173 V=133.3 PL=0
REFP 3 C00174 BC00174
CALL JOB:SEARCH-R1
SET P0305 P0006
SFTON P0305
MOVL C00175 BC00175 V=66.7 PL=0
REFP 3 C00176 BC00176
CALL JOB:SEARCH-R1
SET P0305 P0006
SFTON P0305
MOVL C00177 BC00177 V=66.7 PL=0
SFTOF
'------------------------
'W53A P
'------------------------
SFTOF
MOVJ C00178 BC00178 VJ=30.00
MOVL C00179 BC00179 V=200.0
MOVL C00180 BC00180 V=66.7 PL=0
REFP 3 C00181 BC00181
CALL JOB:SEARCH-R1
SET P0306 P0006
SFTON P0306
MOVL C00182 BC00182 V=66.7 PL=0
REFP 3 C00183 BC00183
CALL JOB:SEARCH-R1
SET P0306 P0006
SFTON P0306
MOVL C00184 BC00184 V=66.7 PL=0
SFTOF
'------------------------
'W56A L
'------------------------
SFTOF
MOVJ C00185 BC00185 VJ=30.00
MOVL C00186 BC00186 V=133.3 PL=0
REFP 3 C00187 BC00187
CALL JOB:SEARCH-R1
SET P0307 P0006
SFTON P0307
MOVL C00188 BC00188 V=66.7 PL=0
REFP 3 C00189 BC00189
CALL JOB:SEARCH-R1
SET P0307 P0006
SFTON P0307
MOVL C00190 BC00190 V=66.7 PL=0
SFTOF
'------------------------
'W56A P
'------------------------
SFTOF
MOVJ C00191 BC00191 VJ=30.00
MOVL C00192 BC00192 V=133.3 PL=0
REFP 3 C00193 BC00193
CALL JOB:SEARCH-R1
SET P0308 P0006
SFTON P0308
MOVL C00194 BC00194 V=66.7 PL=0
REFP 3 C00195 BC00195
CALL JOB:SEARCH-R1
SET P0308 P0006
SFTON P0308
MOVL C00196 BC00196 V=66.7 PL=0
SFTOF
'------------------------
'W52A L
'------------------------
SFTOF
MOVJ C00197 BC00197 VJ=30.00
MOVL C00198 BC00198 V=250.0
MOVL C00199 BC00199 V=66.7 PL=0
REFP 3 C00200 BC00200
CALL JOB:SEARCH-R1
SET P0309 P0006
SFTON P0309
MOVL C00201 BC00201 V=66.7 PL=0
REFP 3 C00202 BC00202
CALL JOB:SEARCH-R1
SET P0309 P0006
SFTON P0309
MOVL C00203 BC00203 V=66.7 PL=0
SFTOF
'------------------------
'W52A P
'------------------------
SFTOF
MOVJ C00204 BC00204 VJ=5.00
MOVJ C00205 BC00205 VJ=20.00
MOVL C00206 BC00206 V=116.7 PL=0
REFP 3 C00207 BC00207
CALL JOB:SEARCH-R1
SET P0310 P0006
SFTON P0310
MOVL C00208 BC00208 V=66.7 PL=0
REFP 3 C00209 BC00209
CALL JOB:SEARCH-R1
SET P0310 P0006
SFTON P0310
MOVL C00210 BC00210 V=66.7 PL=0
SFTOF
'------------------------
'W55A L
'------------------------
SFTOF
MOVL C00211 BC00211 V=250.0
MOVJ C00212 BC00212 VJ=10.00
MOVL C00213 BC00213 V=66.7 PL=0
REFP 3 C00214 BC00214
CALL JOB:SEARCH-R1
SET P0311 P0006
SFTON P0311
MOVL C00215 BC00215 V=66.7 PL=0
REFP 3 C00216 BC00216
CALL JOB:SEARCH-R1
SET P0311 P0006
SFTON P0311
MOVL C00217 BC00217 V=66.7 PL=0
SFTOF
'------------------------
'W55A P
'------------------------
SFTOF
MOVL C00218 BC00218 V=250.0
MOVL C00219 BC00219 V=166.7
MOVL C00220 BC00220 V=66.7 PL=0
REFP 3 C00221 BC00221
CALL JOB:SEARCH-R1
SET P0312 P0006
SFTON P0312
MOVL C00222 BC00222 V=66.7 PL=0
REFP 3 C00223 BC00223
CALL JOB:SEARCH-R1
SET P0312 P0006
SFTON P0312
MOVL C00224 BC00224 V=166.7 PL=0
MOVL C00225 BC00225 V=333.3
SFTOF
MOVL C00226 BC00226 V=333.3
MOVJ C00227 BC00227 VJ=30.00
MOVJ C00228 BC00228 VJ=30.00
MOVJ C00229 BC00229 VJ=20.00
MOVJ C00230 BC00230 VJ=30.00
MOVJ C00231 BC00231 VJ=20.00
MOVJ C00232 BC00232 VJ=20.00
'------------------------
'------------------------
'LEWA STRONA PROFIL GORA
'------------------------
'------------------------
MOVJ C00233 BC00233 VJ=10.00
'------------------------
'W55B L
'------------------------
SFTOF
MOVJ C00234 BC00234 VJ=10.00
MOVL C00235 BC00235 V=166.7 PL=0
REFP 3 C00236 BC00236
CALL JOB:SEARCH-R1
SET P0349 P0006
SFTON P0349
MOVL C00237 BC00237 V=66.7 PL=0
REFP 3 C00238 BC00238
CALL JOB:SEARCH-R1
SET P0349 P0006
SFTON P0349
MOVL C00239 BC00239 V=166.7 PL=0
SFTOF
MOVJ C00240 BC00240 VJ=10.00
MOVJ C00241 BC00241 VJ=20.00
'------------------------
'W55B P
'------------------------
SFTOF
MOVL C00242 BC00242 V=166.7 PL=0
REFP 3 C00243 BC00243
CALL JOB:SEARCH-R1
SET P0350 P0006
SFTON P0350
MOVL C00244 BC00244 V=166.7 PL=0
REFP 3 C00245 BC00245
CALL JOB:SEARCH-R1
SET P0350 P0006
SFTON P0350
MOVL C00246 BC00246 V=166.7 PL=0
SFTOF
'------------------------
'W52B L
'------------------------
SFTOF
MOVJ C00247 BC00247 VJ=20.00
MOVJ C00248 BC00248 VJ=20.00
MOVJ C00249 BC00249 VJ=20.00
MOVL C00250 BC00250 V=150.0
MOVL C00251 BC00251 V=166.7 PL=0
REFP 3 C00252 BC00252
CALL JOB:SEARCH-R1
SET P0351 P0006
SFTON P0351
MOVL C00253 BC00253 V=166.7 PL=0
REFP 3 C00254 BC00254
CALL JOB:SEARCH-R1
SET P0351 P0006
SFTON P0351
MOVL C00255 BC00255 V=166.7 PL=0
SFTOF
'------------------------
'W52B P
'------------------------
SFTOF
MOVJ C00256 BC00256 VJ=30.00
MOVL C00257 BC00257 V=166.7 PL=0
REFP 3 C00258 BC00258
CALL JOB:SEARCH-R1
SET P0352 P0006
SFTON P0352
MOVL C00259 BC00259 V=166.7 PL=0
REFP 3 C00260 BC00260
CALL JOB:SEARCH-R1
SET P0352 P0006
SFTON P0352
MOVL C00261 BC00261 V=166.7 PL=0
SFTOF
'------------------------
'W56B L
'------------------------
SFTOF
MOVJ C00262 BC00262 VJ=30.00
MOVL C00263 BC00263 V=166.7 PL=0
REFP 3 C00264 BC00264
CALL JOB:SEARCH-R1
SET P0353 P0006
SFTON P0353
MOVL C00265 BC00265 V=166.7 PL=0
REFP 3 C00266 BC00266
CALL JOB:SEARCH-R1
SET P0353 P0006
SFTON P0353
MOVL C00267 BC00267 V=166.7 PL=0
SFTOF
'------------------------
'W56B P
'------------------------
SFTOF
MOVJ C00268 BC00268 VJ=30.00
MOVL C00269 BC00269 V=166.7 PL=0
REFP 3 C00270 BC00270
CALL JOB:SEARCH-R1
SET P0354 P0006
SFTON P0354
MOVL C00271 BC00271 V=66.7 PL=0
REFP 3 C00272 BC00272
CALL JOB:SEARCH-R1
SET P0354 P0006
SFTON P0354
MOVL C00273 BC00273 V=66.7 PL=0
SFTOF
'------------------------
'W53B L
'------------------------
SFTOF
MOVJ C00274 BC00274 VJ=30.00
MOVL C00275 BC00275 V=166.7 PL=0
REFP 3 C00276 BC00276
CALL JOB:SEARCH-R1
SET P0355 P0006
SFTON P0355
MOVL C00277 BC00277 V=166.7 PL=0
REFP 3 C00278 BC00278
CALL JOB:SEARCH-R1
SET P0355 P0006
SFTON P0355
MOVL C00279 BC00279 V=166.7 PL=0
SFTOF
'------------------------
'W53B P
'------------------------
SFTOF
MOVJ C00280 BC00280 VJ=30.00
MOVL C00281 BC00281 V=166.7 PL=0
REFP 3 C00282 BC00282
CALL JOB:SEARCH-R1
SET P0356 P0006
SFTON P0356
MOVL C00283 BC00283 V=166.7 PL=0
REFP 3 C00284 BC00284
CALL JOB:SEARCH-R1
SET P0356 P0006
SFTON P0356
MOVL C00285 BC00285 V=166.7 PL=0
SFTOF
'------------------------
'W50B L
'------------------------
SFTOF
MOVJ C00286 BC00286 VJ=30.00
MOVL C00287 BC00287 V=166.7 PL=0
REFP 3 C00288 BC00288
CALL JOB:SEARCH-R1
SET P0357 P0006
SFTON P0357
MOVL C00289 BC00289 V=166.7 PL=0
REFP 3 C00290 BC00290
CALL JOB:SEARCH-R1
SET P0357 P0006
SFTON P0357
MOVL C00291 BC00291 V=166.7 PL=0
SFTOF
'------------------------
'W50B P
'------------------------
SFTOF
MOVJ C00292 BC00292 VJ=30.00
MOVL C00293 BC00293 V=166.7 PL=0
REFP 3 C00294 BC00294
CALL JOB:SEARCH-R1
SET P0358 P0006
SFTON P0358
MOVL C00295 BC00295 V=166.7 PL=0
REFP 3 C00296 BC00296
CALL JOB:SEARCH-R1
SET P0358 P0006
SFTON P0358
MOVL C00297 BC00297 V=166.7 PL=0
SFTOF
'------------------------
'W54B L
'------------------------
SFTOF
MOVJ C00298 BC00298 VJ=30.00
MOVL C00299 BC00299 V=166.7 PL=0
REFP 3 C00300 BC00300
CALL JOB:SEARCH-R1
SET P0359 P0006
SFTON P0359
MOVL C00301 BC00301 V=166.7 PL=0
REFP 3 C00302 BC00302
CALL JOB:SEARCH-R1
SET P0359 P0006
SFTON P0359
MOVL C00303 BC00303 V=166.7 PL=0
SFTOF
'------------------------
'W54B P
'------------------------
SFTOF
MOVJ C00304 BC00304 VJ=30.00
MOVL C00305 BC00305 V=166.7 PL=0
REFP 3 C00306 BC00306
CALL JOB:SEARCH-R1
SET P0360 P0006
SFTON P0360
MOVL C00307 BC00307 V=166.7 PL=0
REFP 3 C00308 BC00308
CALL JOB:SEARCH-R1
SET P0360 P0006
SFTON P0360
MOVL C00309 BC00309 V=166.7 PL=0
MOVL C00310 BC00310 V=333.3
SFTOF
MOVL C00311 BC00311 V=166.7 PL=0
REFP 3 C00312 BC00312
CALL JOB:SEARCH-R1
SET P0361 P0006
SFTON P0361
MOVL C00313 BC00313 V=166.7 PL=0
REFP 3 C00314 BC00314
CALL JOB:SEARCH-R1
SET P0361 P0006
SFTON P0361
MOVL C00315 BC00315 V=166.7
MOVL C00316 BC00316 V=166.7
MOVL C00317 BC00317 V=133.3 PL=0
REFP 3 C00318 BC00318
CALL JOB:SEARCH-R1
SET P0361 P0006
SFTON P0361
SFTOF
MOVL C00319 BC00319 V=250.0
MOVL C00320 BC00320 V=250.0
MOVL C00321 BC00321 V=333.3
MOVJ C00322 BC00322 VJ=20.00
'------------------------
'W51B L
'------------------------
MOVJ C00323 BC00323 VJ=30.00
MOVJ C00324 BC00324 VJ=20.00
MOVJ C00325 BC00325 VJ=40.00
'**********************
'**********************
'POCZATEK SPAWANIA BOKI
'**********************
'**********************
MOVJ C00326 BC00326 VJ=30.00
MOVJ C00327 BC00327 VJ=20.00
'**********************
'W50A
'**********************
MOVL C00328 BC00328 V=250.0
SFTON P0304
MOVL C00329 BC00329 V=83.3 PL=0
SFTOF
MACRO1 MJ#(0) ARGF10
ARCON
SFTON P0303
MOVL C00330 BC00330 V=10.8
ARCOF
SFTOF
MOVL C00331 BC00331 V=150.0
'W13B
MOVJ C00332 BC00332 VJ=10.00
MOVJ C00333 BC00333 VJ=20.00
MOVJ C00334 BC00334 VJ=30.00
MOVJ C00335 BC00335 VJ=30.00
MOVJ C00336 BC00336 VJ=30.00
'**********************
'W50B
'**********************
MOVL C00337 BC00337 V=250.0
SFTON P0357
MOVL C00338 BC00338 V=166.7 PL=0
SFTOF
MACRO1 MJ#(0) ARGF10
ARCON
SFTON P0358
MOVL C00339 BC00339 V=10.8
ARCOF
SFTOF
MOVL C00340 BC00340 V=333.3
MOVJ C00341 BC00341 VJ=30.00
MOVJ C00342 BC00342 VJ=20.00
MOVJ C00343 BC00343 VJ=20.00
MOVJ C00344 BC00344 VJ=20.00
'**********************
'W51A
'**********************
MOVL C00345 BC00345 V=333.3
MACRO1 MJ#(0) ARGF14
MOVL C00346 BC00346 V=250.0
SFTON P0299
MOVL C00347 BC00347 V=83.3 PL=0
ARCON
MOVL C00348 BC00348 V=8.3
ARCOF
SFTOF
MOVL C00349 BC00349 V=416.7
MOVJ C00350 BC00350 VJ=30.00
MOVJ C00351 BC00351 VJ=30.00
MOVJ C00352 BC00352 VJ=30.00
MOVJ C00353 BC00353 VJ=30.00
MOVJ C00354 BC00354 VJ=30.00
MOVJ C00355 BC00355 VJ=30.00
MOVL C00356 BC00356 V=333.3
SFTON P0361
MOVL C00357 BC00357 V=133.3 PL=0
ARCON
MOVL C00358 BC00358 V=8.3
ARCOF
SFTOF
MOVL C00359 BC00359 V=333.3
MOVL C00360 BC00360 V=333.3
MOVJ C00361 BC00361 VJ=30.00
MOVJ C00362 BC00362 VJ=30.00
MOVJ C00363 BC00363 VJ=30.00
MOVJ C00364 BC00364 VJ=40.00
MOVJ C00365 BC00365 VJ=40.00
MOVJ C00366 BC00366 VJ=20.00
MOVJ C00367 BC00367 VJ=20.00
MOVJ C00368 BC00368 VJ=20.00
MOVJ C00369 BC00369 VJ=20.00
MOVJ C00370 BC00370 VJ=20.00
'**********************
'W52A
'**********************
SFTON P0310
MOVL C00371 BC00371 V=250.0
MOVL C00372 BC00372 V=250.0 PL=0
SFTOF
MACRO1 MJ#(0) ARGF10
ARCON
SFTON P0309
MOVL C00373 BC00373 V=10.8
ARCOF
SFTOF
MOVL C00374 BC00374 V=333.3
MOVJ C00375 BC00375 VJ=30.00
MOVJ C00376 BC00376 VJ=30.00
MOVJ C00377 BC00377 VJ=30.00
MOVJ C00378 BC00378 VJ=30.00
MOVJ C00379 BC00379 VJ=30.00
MOVJ C00380 BC00380 VJ=20.00
MOVJ C00381 BC00381 VJ=20.00
MOVJ C00382 BC00382 VJ=20.00
'**********************
'52B
'**********************
MOVL C00383 BC00383 V=250.0
SFTON P0351
MOVL C00384 BC00384 V=83.3 PL=0
SFTOF
MACRO1 MJ#(0) ARGF10
ARCON
SFTON P0352
MOVL C00385 BC00385 V=10.8
ARCOF
MOVL C00386 BC00386 V=333.3
SFTOF
MOVJ C00387 BC00387 VJ=20.00
MOVJ C00388 BC00388 VJ=30.00
MOVJ C00389 BC00389 VJ=30.00
'**********************
'W53A
'**********************
MOVJ C00390 BC00390 VJ=30.00
MOVJ C00391 BC00391 VJ=30.00
MOVJ C00392 BC00392 VJ=10.00
'**********************
'W53A
'**********************
SFTON P0306
MOVL C00393 BC00393 V=250.0
MOVL C00394 BC00394 V=83.3 PL=0
SFTOF
MACRO1 MJ#(0) ARGF10
ARCON
SFTON P0305
MOVL C00395 BC00395 V=10.8
ARCOF
SFTOF
MOVL C00396 BC00396 V=250.0
MOVJ C00397 BC00397 VJ=30.00
MOVJ C00398 BC00398 VJ=30.00
MOVJ C00399 BC00399 VJ=30.00
MOVJ C00400 BC00400 VJ=30.00
MOVJ C00401 BC00401 VJ=30.00
MOVJ C00402 BC00402 VJ=30.00
MOVL C00403 BC00403 V=250.0
'**********************
'W53B
'**********************
SFTON P0351
MOVL C00404 BC00404 V=250.0
MOVL C00405 BC00405 V=166.7 PL=0
SFTOF
MACRO1 MJ#(0) ARGF10
ARCON
SFTON P0350
MOVL C00406 BC00406 V=10.8
ARCOF
SFTOF
MOVL C00407 BC00407 V=333.3
MOVJ C00408 BC00408 VJ=30.00
MOVJ C00409 BC00409 VJ=30.00
MOVJ C00410 BC00410 VJ=30.00
MOVJ C00411 BC00411 VJ=30.00
MOVJ C00412 BC00412 VJ=30.00
'**********************
'W54A
'**********************
SFTON P0302
MOVL C00413 BC00413 V=250.0
MOVL C00414 BC00414 V=83.3 PL=0
SFTOF
MACRO1 MJ#(0) ARGF10
ARCON
SFTON P0301
MOVL C00415 BC00415 V=10.8
ARCOF
SFTOF
MOVL C00416 BC00416 V=333.3
MOVJ C00417 BC00417 VJ=20.00
MOVJ C00418 BC00418 VJ=30.00
MOVJ C00419 BC00419 VJ=30.00
MOVJ C00420 BC00420 VJ=30.00
MOVJ C00421 BC00421 VJ=30.00
'**********************
'W54B
'**********************
SFTON P0359
MOVL C00422 BC00422 V=416.7
MOVL C00423 BC00423 V=166.7 PL=0
SFTOF
MACRO1 MJ#(0) ARGF10
ARCON
SFTON P0360
MOVL C00424 BC00424 V=10.8
ARCOF
MOVL C00425 BC00425 V=333.3
SFTOF
MOVJ C00426 BC00426 VJ=30.00
MOVJ C00427 BC00427 VJ=40.00
MOVJ C00428 BC00428 VJ=30.00
MOVJ C00429 BC00429 VJ=40.00
MOVJ C00430 BC00430 VJ=40.00
MOVJ C00431 BC00431 VJ=10.00
MOVJ C00432 BC00432 VJ=15.00
MOVJ C00433 BC00433 VJ=10.00
MOVJ C00434 BC00434 VJ=10.00
MOVJ C00435 BC00435 VJ=10.00
MOVJ C00436 BC00436 VJ=10.00
MOVJ C00437 BC00437 VJ=10.00
'**********************
'W55A
'**********************
SFTON P0311
MOVL C00438 BC00438 V=166.7 PL=0
SFTOF
MACRO1 MJ#(0) ARGF10
ARCON
SFTON P0312
MOVL C00439 BC00439 V=10.8
MOVL C00440 BC00440 V=10.8
ARCOF
SFTOF
MOVL C00441 BC00441 V=150.0
MOVJ C00442 BC00442 VJ=10.00
MOVJ C00443 BC00443 VJ=10.00
MOVJ C00444 BC00444 VJ=10.00
MOVJ C00445 BC00445 VJ=10.00
MOVJ C00446 BC00446 VJ=10.00
MOVJ C00447 BC00447 VJ=10.00
MOVJ C00448 BC00448 VJ=15.00
MOVJ C00449 BC00449 VJ=15.00
MOVJ C00450 BC00450 VJ=20.00
MOVJ C00451 BC00451 VJ=20.00
MOVJ C00452 BC00452 VJ=20.00
MOVJ C00453 BC00453 VJ=20.00
MOVJ C00454 BC00454 VJ=20.00
MOVJ C00455 BC00455 VJ=10.00
MOVJ C00456 BC00456 VJ=10.00
'**********************
'W55B
'**********************
SFTON P0350
MOVL C00457 BC00457 V=166.7
MOVL C00458 BC00458 V=83.3 PL=0
SFTOF
MACRO1 MJ#(0) ARGF10
ARCON
SFTON P0349
MOVL C00459 BC00459 V=10.8
MOVL C00460 BC00460 V=10.8
ARCOF
SFTOF
MOVL C00461 BC00461 V=166.7
MOVJ C00462 BC00462 VJ=10.00
MOVJ C00463 BC00463 VJ=10.00
MOVJ C00464 BC00464 VJ=10.00
MOVJ C00465 BC00465 VJ=10.00
MOVJ C00466 BC00466 VJ=10.00
MOVJ C00467 BC00467 VJ=30.00
MOVJ C00468 BC00468 VJ=30.00
MOVJ C00469 BC00469 VJ=30.00
MOVJ C00470 BC00470 VJ=20.00
'**********************
'W56A
'**********************
SFTON P0308
MOVL C00471 BC00471 V=166.7
MOVL C00472 BC00472 V=83.3 PL=0
SFTOF
MACRO1 MJ#(0) ARGF10
ARCON
SFTON P0307
MOVL C00473 BC00473 V=10.8
ARCOF
SFTOF
MOVL C00474 BC00474 V=333.3
MOVJ C00475 BC00475 VJ=20.00
MOVJ C00476 BC00476 VJ=30.00
MOVJ C00477 BC00477 VJ=30.00
MOVJ C00478 BC00478 VJ=30.00
'**********************
'W56B
'**********************
SFTON P0353
MOVL C00479 BC00479 V=250.0
MOVL C00480 BC00480 V=166.7 PL=0
SFTOF
MACRO1 MJ#(0) ARGF10
ARCON
SFTON P0354
MOVL C00481 BC00481 V=10.8
ARCOF
SFTOF
MOVL C00482 BC00482 V=333.3
MOVJ C00483 BC00483 VJ=30.00
MOVJ C00484 BC00484 VJ=30.00
MOVJ C00485 BC00485 VJ=30.00
CALL JOB:MOVE_OUT_OF_TUNNEL
CALL JOB:R1-HOME
END
